FUNCTION_BLOCK PushControl (* Basic Function Block Type *)
  (* Standard: 61499-2 *)
  (* Version 0.0, 22/06/2022, Lernfabrik, WBK hackaton, Template *)
  PACKAGE Main;
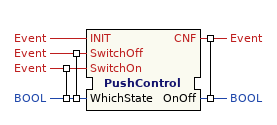
  EVENT_INPUT
    INIT; (* Initialization Request *)
    SwitchOff WITH WhichState;
    SwitchOn WITH WhichState;
  END_EVENT
  EVENT_OUTPUT
    CNF WITH OnOff; (* Execution Confirmation *)
  END_EVENT
  VAR_INPUT
    WhichState : BOOL;
  END_VAR
  VAR_OUTPUT
    OnOff : BOOL; (* Output event qualifier *)
  END_VAR
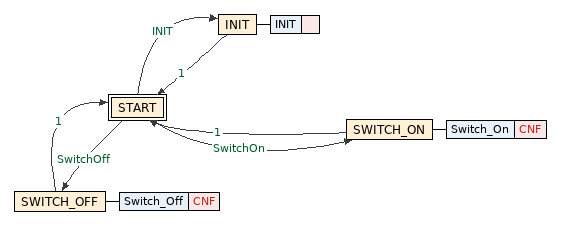
  EC_STATES
    START; (* Initial State *)
    INIT : INIT; (* Initialization *)
    SWITCH_OFF : Switch_Off -> CNF; (* Normal execution *)
    SWITCH_ON : Switch_On -> CNF;
  END_STATES
  EC_TRANSITIONS
    START TO INIT := INIT;
    INIT TO START := 1;
    START TO SWITCH_OFF := SwitchOff;
    SWITCH_OFF TO START := 1;
    START TO SWITCH_ON := SwitchOn;
    SWITCH_ON TO START := 1;
  END_TRANSITIONS
  ALGORITHM INIT IN ST: (* Initialization algorithm *)
OnOff := 0;
  END_ALGORITHM
  ALGORITHM REQ IN ST: (* Normally executed algorithm *)
;
  END_ALGORITHM
  ALGORITHM Switch_Off IN ST:
OnOff := 0;
  END_ALGORITHM
  ALGORITHM Switch_On IN ST:
OnOff := 1;
  END_ALGORITHM
END_FUNCTION_BLOCK
